Fanuc KAREL source: SET_CURSOR.kl

PROGRAM T
%NOLOCKGROUP
VAR
 v0 : FILE
 v1 : INTEGER
 v2 : INTEGER
 v3 : INTEGER
BEGIN
 SET_CURSOR(v0, v1, v2, v3)
END T
